TYPE U_SDO_DATA :
UNION
	aData : ARRAY[0..3] OF BYTE;
	nData : DINT;
	sData : STRING(20);
END_UNION
END_TYPE

(* stored: Version 1.1.0.1, ProductVersion 3.1.0.25
   DUT U_SDO_DATA: Id {695f0b1e-a409-47b7-941b-b05041a79c28} *)
